// TIA Portal V17 export
// export: Created 2023-04-03T06:31:26.4990161Z, ExportSetting WithDefaults, DisplayName Totally Integrated Automation Portal, DisplayVersion V17 Update 4, DisplayName TIA Portal Openness, DisplayVersion V17 Update 4, DisplayName TIA Portal Version Control Interface, DisplayVersion V17, DisplayName STEP 7 Professional, DisplayVersion V17 Update 4, DisplayName STEP 7 Safety, DisplayVersion V17, DisplayName WinCC Professional, DisplayVersion V17 Update 4
FUNCTION "PCS R (F)_1" : Void   // FC47, LAD
TITLE = ModBus TCP for PCS Power Electronics
{ S7_Optimized_Access := 'TRUE' }
VERSION : 0.1
// stored: AutoNumber true, IsIECCheckEnabled false, SetENOAutomatically false, UDAEnableTagReadback false
   VAR_TEMP
      rVac : Real;
   END_VAR
   VAR_TEMP   // added for the SCL form of the ladder/FBD networks
      _w1 : Bool;
   END_VAR
BEGIN

REGION Network 1: Function Modbus Client 10
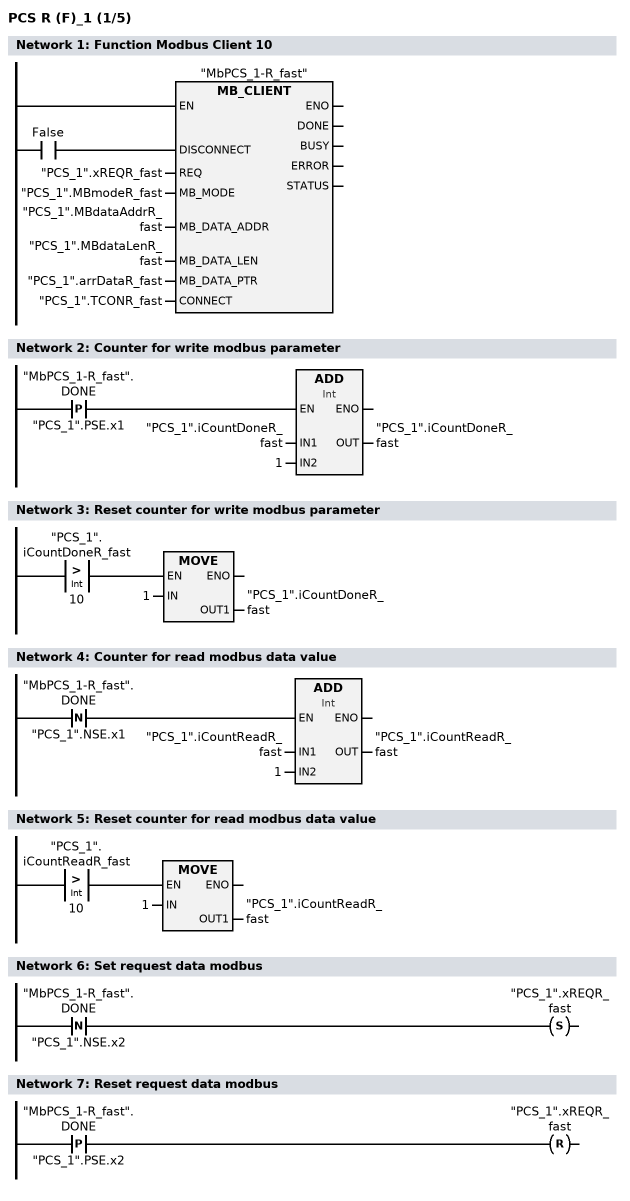
   RUNG wire#powerrail
      "MbPCS_1-R_fast".MB_CLIENT(DISCONNECT := wire#w1, REQ := "PCS_1".xREQR_fast, MB_MODE := "PCS_1".MBmodeR_fast, MB_DATA_ADDR := "PCS_1".MBdataAddrR_fast, MB_DATA_LEN := "PCS_1".MBdataLenR_fast, MB_DATA_PTR := "PCS_1".arrDataR_fast, CONNECT := "PCS_1".TCONR_fast, DONE =>, BUSY =>, ERROR =>, STATUS =>)
   END_RUNG
   RUNG wire#powerrail
      Contact( False )
   END_RUNG wire#w1
   // the same network as SCL:
   "MbPCS_1-R_fast"(DISCONNECT := False,   // MB_CLIENT
                    REQ := "PCS_1".xREQR_fast,
                    MB_MODE := "PCS_1".MBmodeR_fast,
                    MB_DATA_ADDR := "PCS_1".MBdataAddrR_fast,
                    MB_DATA_LEN := "PCS_1".MBdataLenR_fast,
                    MB_DATA_PTR := "PCS_1".arrDataR_fast,
                    CONNECT := "PCS_1".TCONR_fast);
END_REGION

REGION Network 2: Counter for write modbus parameter
   RUNG wire#powerrail
      P_Contact(operand := "MbPCS_1-R_fast".DONE, bit := "PCS_1".PSE.x1)
      { S7_Templates := "SrcType := Int" } Add(in1 := "PCS_1".iCountDoneR_fast, in2 := 1, out => "PCS_1".iCountDoneR_fast)
   END_RUNG
   // the same network as SCL:
   #_w1 := "MbPCS_1-R_fast".DONE AND NOT "PCS_1".PSE.x1;   // rising edge of "MbPCS_1-R_fast".DONE
   "PCS_1".PSE.x1 := "MbPCS_1-R_fast".DONE;
   IF #_w1 THEN "PCS_1".iCountDoneR_fast := "PCS_1".iCountDoneR_fast + 1; END_IF;
END_REGION

REGION Network 3: Reset counter for write modbus parameter
   RUNG wire#powerrail
      { S7_Templates := "SrcType := Int" } GT_Contact(in1 := "PCS_1".iCountDoneR_fast, in2 := 10)
      Move(in := 1, out1 => "PCS_1".iCountDoneR_fast)
   END_RUNG
   // the same network as SCL:
   IF "PCS_1".iCountDoneR_fast > 10 THEN "PCS_1".iCountDoneR_fast := 1; END_IF;
END_REGION

REGION Network 4: Counter for read modbus data value
   RUNG wire#powerrail
      N_Contact(operand := "MbPCS_1-R_fast".DONE, bit := "PCS_1".NSE.x1)
      { S7_Templates := "SrcType := Int" } Add(in1 := "PCS_1".iCountReadR_fast, in2 := 1, out => "PCS_1".iCountReadR_fast)
   END_RUNG
   // the same network as SCL:
   #_w1 := NOT "MbPCS_1-R_fast".DONE AND "PCS_1".NSE.x1;   // falling edge of "MbPCS_1-R_fast".DONE
   "PCS_1".NSE.x1 := "MbPCS_1-R_fast".DONE;
   IF #_w1 THEN "PCS_1".iCountReadR_fast := "PCS_1".iCountReadR_fast + 1; END_IF;
END_REGION

REGION Network 5: Reset counter for read modbus data value
   RUNG wire#powerrail
      { S7_Templates := "SrcType := Int" } GT_Contact(in1 := "PCS_1".iCountReadR_fast, in2 := 10)
      Move(in := 1, out1 => "PCS_1".iCountReadR_fast)
   END_RUNG
   // the same network as SCL:
   IF "PCS_1".iCountReadR_fast > 10 THEN "PCS_1".iCountReadR_fast := 1; END_IF;
END_REGION

REGION Network 6: Set request data modbus
   RUNG wire#powerrail
      N_Contact(operand := "MbPCS_1-R_fast".DONE, bit := "PCS_1".NSE.x2)
      S_Coil( "PCS_1".xREQR_fast )
   END_RUNG
   // the same network as SCL:
   #_w1 := NOT "MbPCS_1-R_fast".DONE AND "PCS_1".NSE.x2;   // falling edge of "MbPCS_1-R_fast".DONE
   "PCS_1".NSE.x2 := "MbPCS_1-R_fast".DONE;
   IF #_w1 THEN "PCS_1".xREQR_fast := TRUE; END_IF;
END_REGION

REGION Network 7: Reset request data modbus
   RUNG wire#powerrail
      P_Contact(operand := "MbPCS_1-R_fast".DONE, bit := "PCS_1".PSE.x2)
      R_Coil( "PCS_1".xREQR_fast )
   END_RUNG
   // the same network as SCL:
   #_w1 := "MbPCS_1-R_fast".DONE AND NOT "PCS_1".PSE.x2;   // rising edge of "MbPCS_1-R_fast".DONE
   "PCS_1".PSE.x2 := "MbPCS_1-R_fast".DONE;
   IF #_w1 THEN "PCS_1".xREQR_fast := FALSE; END_IF;
END_REGION

REGION Network 8: Write R_Block1 parameter - new
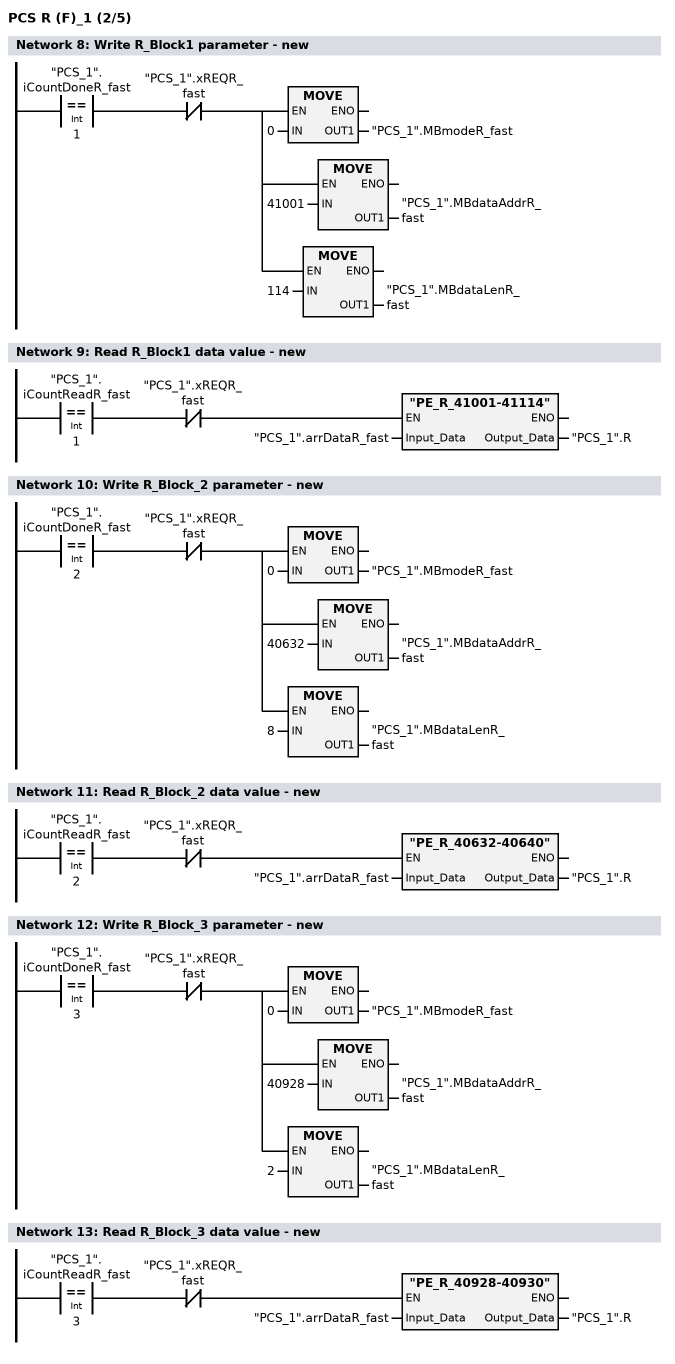
   RUNG wire#powerrail
      { S7_Templates := "SrcType := Int" } EQ_Contact(in1 := "PCS_1".iCountDoneR_fast, in2 := 1)
      I_Contact( "PCS_1".xREQR_fast )
      wire#w1
      Move(in := 0, out1 => "PCS_1".MBmodeR_fast)
   END_RUNG
   RUNG wire#w1
      Move(in := 41001, out1 => "PCS_1".MBdataAddrR_fast)
   END_RUNG
   RUNG wire#w1
      Move(in := 114, out1 => "PCS_1".MBdataLenR_fast)
   END_RUNG
   // the same network as SCL:
   IF ("PCS_1".iCountDoneR_fast = 1) AND NOT "PCS_1".xREQR_fast THEN
       "PCS_1".MBmodeR_fast := 0;
       "PCS_1".MBdataAddrR_fast := 41001;
       "PCS_1".MBdataLenR_fast := 114;
   END_IF;
END_REGION

REGION Network 9: Read R_Block1 data value - new
   RUNG wire#powerrail
      { S7_Templates := "SrcType := Int" } EQ_Contact(in1 := "PCS_1".iCountReadR_fast, in2 := 1)
      I_Contact( "PCS_1".xREQR_fast )
      "PE_R_41001-41114"(Input_Data := "PCS_1".arrDataR_fast, Output_Data => "PCS_1".R)
   END_RUNG
   // the same network as SCL:
   IF ("PCS_1".iCountReadR_fast = 1) AND NOT "PCS_1".xREQR_fast THEN
       "PE_R_41001-41114"(Input_Data := "PCS_1".arrDataR_fast, Output_Data => "PCS_1".R);
   END_IF;
END_REGION

REGION Network 10: Write R_Block_2 parameter - new
   RUNG wire#powerrail
      { S7_Templates := "SrcType := Int" } EQ_Contact(in1 := "PCS_1".iCountDoneR_fast, in2 := 2)
      I_Contact( "PCS_1".xREQR_fast )
      wire#w1
      Move(in := 0, out1 => "PCS_1".MBmodeR_fast)
   END_RUNG
   RUNG wire#w1
      Move(in := 40632, out1 => "PCS_1".MBdataAddrR_fast)
   END_RUNG
   RUNG wire#w1
      Move(in := 8, out1 => "PCS_1".MBdataLenR_fast)
   END_RUNG
   // the same network as SCL:
   IF ("PCS_1".iCountDoneR_fast = 2) AND NOT "PCS_1".xREQR_fast THEN
       "PCS_1".MBmodeR_fast := 0;
       "PCS_1".MBdataAddrR_fast := 40632;
       "PCS_1".MBdataLenR_fast := 8;
   END_IF;
END_REGION

REGION Network 11: Read R_Block_2 data value - new
   RUNG wire#powerrail
      { S7_Templates := "SrcType := Int" } EQ_Contact(in1 := "PCS_1".iCountReadR_fast, in2 := 2)
      I_Contact( "PCS_1".xREQR_fast )
      "PE_R_40632-40640"(Input_Data := "PCS_1".arrDataR_fast, Output_Data => "PCS_1".R)
   END_RUNG
   // the same network as SCL:
   IF ("PCS_1".iCountReadR_fast = 2) AND NOT "PCS_1".xREQR_fast THEN
       "PE_R_40632-40640"(Input_Data := "PCS_1".arrDataR_fast, Output_Data => "PCS_1".R);
   END_IF;
END_REGION

REGION Network 12: Write R_Block_3 parameter - new
   RUNG wire#powerrail
      { S7_Templates := "SrcType := Int" } EQ_Contact(in1 := "PCS_1".iCountDoneR_fast, in2 := 3)
      I_Contact( "PCS_1".xREQR_fast )
      wire#w1
      Move(in := 0, out1 => "PCS_1".MBmodeR_fast)
   END_RUNG
   RUNG wire#w1
      Move(in := 40928, out1 => "PCS_1".MBdataAddrR_fast)
   END_RUNG
   RUNG wire#w1
      Move(in := 2, out1 => "PCS_1".MBdataLenR_fast)
   END_RUNG
   // the same network as SCL:
   IF ("PCS_1".iCountDoneR_fast = 3) AND NOT "PCS_1".xREQR_fast THEN
       "PCS_1".MBmodeR_fast := 0;
       "PCS_1".MBdataAddrR_fast := 40928;
       "PCS_1".MBdataLenR_fast := 2;
   END_IF;
END_REGION

REGION Network 13: Read R_Block_3 data value - new
   RUNG wire#powerrail
      { S7_Templates := "SrcType := Int" } EQ_Contact(in1 := "PCS_1".iCountReadR_fast, in2 := 3)
      I_Contact( "PCS_1".xREQR_fast )
      "PE_R_40928-40930"(Input_Data := "PCS_1".arrDataR_fast, Output_Data => "PCS_1".R)
   END_RUNG
   // the same network as SCL:
   IF ("PCS_1".iCountReadR_fast = 3) AND NOT "PCS_1".xREQR_fast THEN
       "PE_R_40928-40930"(Input_Data := "PCS_1".arrDataR_fast, Output_Data => "PCS_1".R);
   END_IF;
END_REGION

REGION Network 14: Write R_Block_4 parameter - new
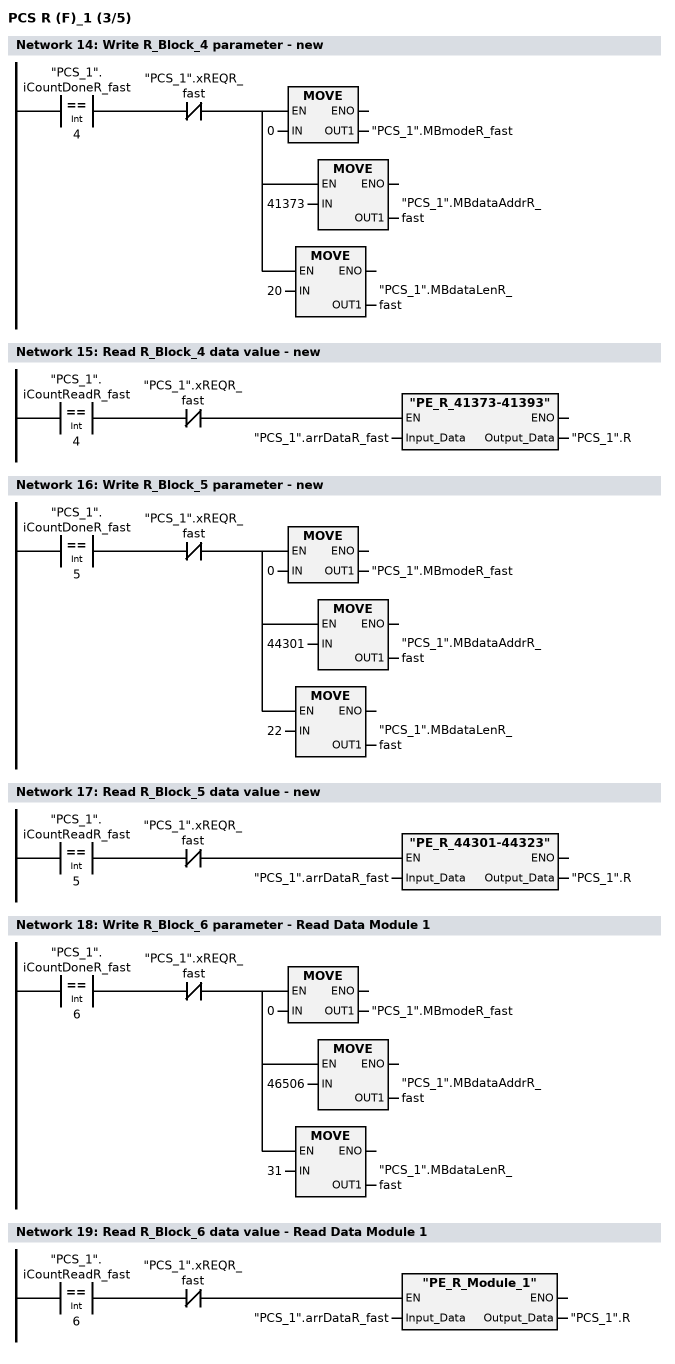
   RUNG wire#powerrail
      { S7_Templates := "SrcType := Int" } EQ_Contact(in1 := "PCS_1".iCountDoneR_fast, in2 := 4)
      I_Contact( "PCS_1".xREQR_fast )
      wire#w1
      Move(in := 0, out1 => "PCS_1".MBmodeR_fast)
   END_RUNG
   RUNG wire#w1
      Move(in := 41373, out1 => "PCS_1".MBdataAddrR_fast)
   END_RUNG
   RUNG wire#w1
      Move(in := 20, out1 => "PCS_1".MBdataLenR_fast)
   END_RUNG
   // the same network as SCL:
   IF ("PCS_1".iCountDoneR_fast = 4) AND NOT "PCS_1".xREQR_fast THEN
       "PCS_1".MBmodeR_fast := 0;
       "PCS_1".MBdataAddrR_fast := 41373;
       "PCS_1".MBdataLenR_fast := 20;
   END_IF;
END_REGION

REGION Network 15: Read R_Block_4 data value - new
   RUNG wire#powerrail
      { S7_Templates := "SrcType := Int" } EQ_Contact(in1 := "PCS_1".iCountReadR_fast, in2 := 4)
      I_Contact( "PCS_1".xREQR_fast )
      "PE_R_41373-41393"(Input_Data := "PCS_1".arrDataR_fast, Output_Data => "PCS_1".R)
   END_RUNG
   // the same network as SCL:
   IF ("PCS_1".iCountReadR_fast = 4) AND NOT "PCS_1".xREQR_fast THEN
       "PE_R_41373-41393"(Input_Data := "PCS_1".arrDataR_fast, Output_Data => "PCS_1".R);
   END_IF;
END_REGION

REGION Network 16: Write R_Block_5 parameter - new
   RUNG wire#powerrail
      { S7_Templates := "SrcType := Int" } EQ_Contact(in1 := "PCS_1".iCountDoneR_fast, in2 := 5)
      I_Contact( "PCS_1".xREQR_fast )
      wire#w1
      Move(in := 0, out1 => "PCS_1".MBmodeR_fast)
   END_RUNG
   RUNG wire#w1
      Move(in := 44301, out1 => "PCS_1".MBdataAddrR_fast)
   END_RUNG
   RUNG wire#w1
      Move(in := 22, out1 => "PCS_1".MBdataLenR_fast)
   END_RUNG
   // the same network as SCL:
   IF ("PCS_1".iCountDoneR_fast = 5) AND NOT "PCS_1".xREQR_fast THEN
       "PCS_1".MBmodeR_fast := 0;
       "PCS_1".MBdataAddrR_fast := 44301;
       "PCS_1".MBdataLenR_fast := 22;
   END_IF;
END_REGION

REGION Network 17: Read R_Block_5 data value - new
   RUNG wire#powerrail
      { S7_Templates := "SrcType := Int" } EQ_Contact(in1 := "PCS_1".iCountReadR_fast, in2 := 5)
      I_Contact( "PCS_1".xREQR_fast )
      "PE_R_44301-44323"(Input_Data := "PCS_1".arrDataR_fast, Output_Data => "PCS_1".R)
   END_RUNG
   // the same network as SCL:
   IF ("PCS_1".iCountReadR_fast = 5) AND NOT "PCS_1".xREQR_fast THEN
       "PE_R_44301-44323"(Input_Data := "PCS_1".arrDataR_fast, Output_Data => "PCS_1".R);
   END_IF;
END_REGION

REGION Network 18: Write R_Block_6 parameter - Read Data Module 1
   RUNG wire#powerrail
      { S7_Templates := "SrcType := Int" } EQ_Contact(in1 := "PCS_1".iCountDoneR_fast, in2 := 6)
      I_Contact( "PCS_1".xREQR_fast )
      wire#w1
      Move(in := 0, out1 => "PCS_1".MBmodeR_fast)
   END_RUNG
   RUNG wire#w1
      Move(in := 46506, out1 => "PCS_1".MBdataAddrR_fast)
   END_RUNG
   RUNG wire#w1
      Move(in := 31, out1 => "PCS_1".MBdataLenR_fast)
   END_RUNG
   // the same network as SCL:
   IF ("PCS_1".iCountDoneR_fast = 6) AND NOT "PCS_1".xREQR_fast THEN
       "PCS_1".MBmodeR_fast := 0;
       "PCS_1".MBdataAddrR_fast := 46506;
       "PCS_1".MBdataLenR_fast := 31;
   END_IF;
END_REGION

REGION Network 19: Read R_Block_6 data value - Read Data Module 1
   RUNG wire#powerrail
      { S7_Templates := "SrcType := Int" } EQ_Contact(in1 := "PCS_1".iCountReadR_fast, in2 := 6)
      I_Contact( "PCS_1".xREQR_fast )
      "PE_R_Module_1"(Input_Data := "PCS_1".arrDataR_fast, Output_Data => "PCS_1".R)
   END_RUNG
   // the same network as SCL:
   IF ("PCS_1".iCountReadR_fast = 6) AND NOT "PCS_1".xREQR_fast THEN
       "PE_R_Module_1"(Input_Data := "PCS_1".arrDataR_fast, Output_Data => "PCS_1".R);
   END_IF;
END_REGION

REGION Network 20: Write R_Block_7 parameter - Read Data Module 2
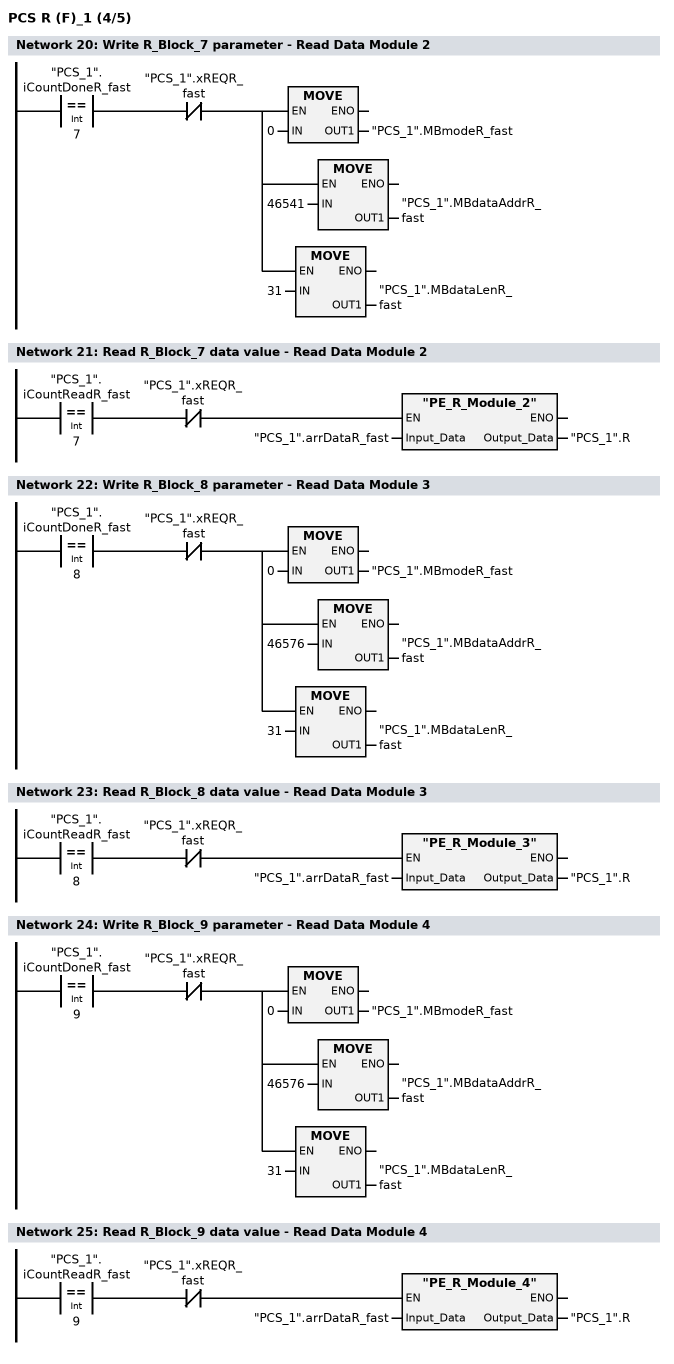
   RUNG wire#powerrail
      { S7_Templates := "SrcType := Int" } EQ_Contact(in1 := "PCS_1".iCountDoneR_fast, in2 := 7)
      I_Contact( "PCS_1".xREQR_fast )
      wire#w1
      Move(in := 0, out1 => "PCS_1".MBmodeR_fast)
   END_RUNG
   RUNG wire#w1
      Move(in := 46541, out1 => "PCS_1".MBdataAddrR_fast)
   END_RUNG
   RUNG wire#w1
      Move(in := 31, out1 => "PCS_1".MBdataLenR_fast)
   END_RUNG
   // the same network as SCL:
   IF ("PCS_1".iCountDoneR_fast = 7) AND NOT "PCS_1".xREQR_fast THEN
       "PCS_1".MBmodeR_fast := 0;
       "PCS_1".MBdataAddrR_fast := 46541;
       "PCS_1".MBdataLenR_fast := 31;
   END_IF;
END_REGION

REGION Network 21: Read R_Block_7 data value - Read Data Module 2
   RUNG wire#powerrail
      { S7_Templates := "SrcType := Int" } EQ_Contact(in1 := "PCS_1".iCountReadR_fast, in2 := 7)
      I_Contact( "PCS_1".xREQR_fast )
      "PE_R_Module_2"(Input_Data := "PCS_1".arrDataR_fast, Output_Data => "PCS_1".R)
   END_RUNG
   // the same network as SCL:
   IF ("PCS_1".iCountReadR_fast = 7) AND NOT "PCS_1".xREQR_fast THEN
       "PE_R_Module_2"(Input_Data := "PCS_1".arrDataR_fast, Output_Data => "PCS_1".R);
   END_IF;
END_REGION

REGION Network 22: Write R_Block_8 parameter - Read Data Module 3
   RUNG wire#powerrail
      { S7_Templates := "SrcType := Int" } EQ_Contact(in1 := "PCS_1".iCountDoneR_fast, in2 := 8)
      I_Contact( "PCS_1".xREQR_fast )
      wire#w1
      Move(in := 0, out1 => "PCS_1".MBmodeR_fast)
   END_RUNG
   RUNG wire#w1
      Move(in := 46576, out1 => "PCS_1".MBdataAddrR_fast)
   END_RUNG
   RUNG wire#w1
      Move(in := 31, out1 => "PCS_1".MBdataLenR_fast)
   END_RUNG
   // the same network as SCL:
   IF ("PCS_1".iCountDoneR_fast = 8) AND NOT "PCS_1".xREQR_fast THEN
       "PCS_1".MBmodeR_fast := 0;
       "PCS_1".MBdataAddrR_fast := 46576;
       "PCS_1".MBdataLenR_fast := 31;
   END_IF;
END_REGION

REGION Network 23: Read R_Block_8 data value - Read Data Module 3
   RUNG wire#powerrail
      { S7_Templates := "SrcType := Int" } EQ_Contact(in1 := "PCS_1".iCountReadR_fast, in2 := 8)
      I_Contact( "PCS_1".xREQR_fast )
      "PE_R_Module_3"(Input_Data := "PCS_1".arrDataR_fast, Output_Data => "PCS_1".R)
   END_RUNG
   // the same network as SCL:
   IF ("PCS_1".iCountReadR_fast = 8) AND NOT "PCS_1".xREQR_fast THEN
       "PE_R_Module_3"(Input_Data := "PCS_1".arrDataR_fast, Output_Data => "PCS_1".R);
   END_IF;
END_REGION

REGION Network 24: Write R_Block_9 parameter - Read Data Module 4
   RUNG wire#powerrail
      { S7_Templates := "SrcType := Int" } EQ_Contact(in1 := "PCS_1".iCountDoneR_fast, in2 := 9)
      I_Contact( "PCS_1".xREQR_fast )
      wire#w1
      Move(in := 0, out1 => "PCS_1".MBmodeR_fast)
   END_RUNG
   RUNG wire#w1
      Move(in := 46576, out1 => "PCS_1".MBdataAddrR_fast)
   END_RUNG
   RUNG wire#w1
      Move(in := 31, out1 => "PCS_1".MBdataLenR_fast)
   END_RUNG
   // the same network as SCL:
   IF ("PCS_1".iCountDoneR_fast = 9) AND NOT "PCS_1".xREQR_fast THEN
       "PCS_1".MBmodeR_fast := 0;
       "PCS_1".MBdataAddrR_fast := 46576;
       "PCS_1".MBdataLenR_fast := 31;
   END_IF;
END_REGION

REGION Network 25: Read R_Block_9 data value - Read Data Module 4
   RUNG wire#powerrail
      { S7_Templates := "SrcType := Int" } EQ_Contact(in1 := "PCS_1".iCountReadR_fast, in2 := 9)
      I_Contact( "PCS_1".xREQR_fast )
      "PE_R_Module_4"(Input_Data := "PCS_1".arrDataR_fast, Output_Data => "PCS_1".R)
   END_RUNG
   // the same network as SCL:
   IF ("PCS_1".iCountReadR_fast = 9) AND NOT "PCS_1".xREQR_fast THEN
       "PE_R_Module_4"(Input_Data := "PCS_1".arrDataR_fast, Output_Data => "PCS_1".R);
   END_IF;
END_REGION

REGION Network 26: Write R_Block_10 parameter - Read Humidity module 1-2-3-4
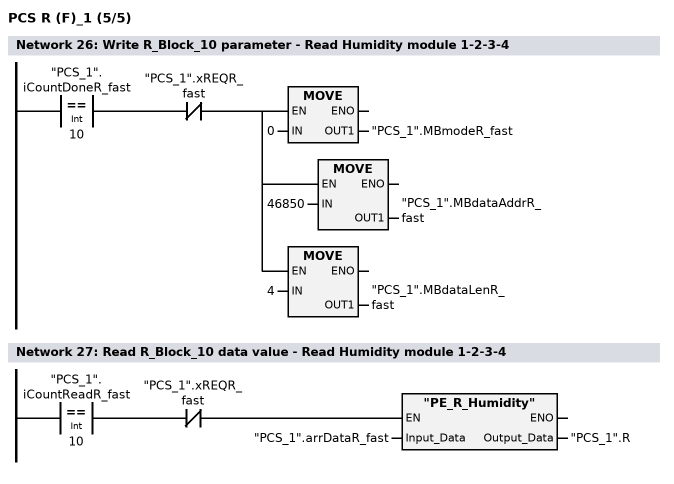
   RUNG wire#powerrail
      { S7_Templates := "SrcType := Int" } EQ_Contact(in1 := "PCS_1".iCountDoneR_fast, in2 := 10)
      I_Contact( "PCS_1".xREQR_fast )
      wire#w1
      Move(in := 0, out1 => "PCS_1".MBmodeR_fast)
   END_RUNG
   RUNG wire#w1
      Move(in := 46850, out1 => "PCS_1".MBdataAddrR_fast)
   END_RUNG
   RUNG wire#w1
      Move(in := 4, out1 => "PCS_1".MBdataLenR_fast)
   END_RUNG
   // the same network as SCL:
   IF ("PCS_1".iCountDoneR_fast = 10) AND NOT "PCS_1".xREQR_fast THEN
       "PCS_1".MBmodeR_fast := 0;
       "PCS_1".MBdataAddrR_fast := 46850;
       "PCS_1".MBdataLenR_fast := 4;
   END_IF;
END_REGION

REGION Network 27: Read R_Block_10 data value - Read Humidity module 1-2-3-4
   RUNG wire#powerrail
      { S7_Templates := "SrcType := Int" } EQ_Contact(in1 := "PCS_1".iCountReadR_fast, in2 := 10)
      I_Contact( "PCS_1".xREQR_fast )
      "PE_R_Humidity"(Input_Data := "PCS_1".arrDataR_fast, Output_Data => "PCS_1".R)
   END_RUNG
   // the same network as SCL:
   IF ("PCS_1".iCountReadR_fast = 10) AND NOT "PCS_1".xREQR_fast THEN
       "PE_R_Humidity"(Input_Data := "PCS_1".arrDataR_fast, Output_Data => "PCS_1".R);
   END_IF;
END_REGION
END_FUNCTION
